// TwinCAT 3 PLC project HardwareSimulator
// ProgramVersion: 3.1.4024.0
// libraries:
//   Tc2_Standard, * (Beckhoff Automation GmbH)
//   Tc2_System, * (Beckhoff Automation GmbH)
//   Tc2_Utilities, * (Beckhoff Automation GmbH)
//   Tc3_Module, * (Beckhoff Automation GmbH)
//   VisuSymbols,3.5.10.0,System
// project tree:
//   / GlobalTextList.TcGTLO (not stored), PlcTask.TcTTO, Visualization Manager.TcVMO (not stored)
//   POUs/ MAIN.TcPOU, SIM_ValveWithFB.TcPOU, SIM_ValveWithDoubleFB.TcPOU, SIM_MOVITRAC_B.TcPOU, SIM_SpeedDoor.TcPOU
//   VISUs/ Visualization.TcVIS
// (motion and I/O tree: see PLC project cleanroomconnect)
// real-time tasks:
//   TASK PlcTask: cycle T#10ms, priority 20, ADS port 350
//   TASK PlcTaskHwSim: cycle T#10ms, priority 21, ADS port 351
// variable links:

CONFIGURATION HardwareSimulator
    RESOURCE PLC ON TwinCAT3
        TASK PlcTask(INTERVAL := T#10ms, PRIORITY := 21);
        PROGRAM MAIN WITH PlcTask : MAIN;
    END_RESOURCE
END_CONFIGURATION

// ---- POUs/MAIN.TcPOU
PROGRAM MAIN
VAR
	//EM Pallet Transport
	simMOVITRAC_B : SIM_MOVITRAC_B;
	simCentering : SIM_ValveWithDoubleFB;
	
	//EM Docking Interface
	simDockingClampUpper : SIM_ValveWithDoubleFB;
	simDockingClampLower : SIM_ValveWithDoubleFB;
	simUnlockPinUpper : SIM_ValveWithFB;
	simUnlockPinLower : SIM_ValveWithFB;
	simDoorOpener : SIM_ValveWithFB;
	simDoorShutter : SIM_ValveWithFB;
	simDoorOpenerAlmostClosed AT %Q* : BOOL;
	tonDoorOpenerAlmosClosed : TON;
	
	//EM Lifting Transport
 	//Via NC-Task
	
	//EM Doors
	simOuterCabinDoor : SIM_SpeedDoor;
	simInnerCabinDoor : SIM_SpeedDoor;
	
	//Safety
	bInitDone : BOOL;
	simSafetyOK AT %Q* : BOOL;
	simPower400VacOK AT %Q* : BOOL;
	simPower230VacOK AT %Q* : BOOL;
	simPower230VacSocketsOK AT %Q* : BOOL;
	simPower48VdcOK AT %Q* : BOOL;
	simPowerPotentialGroupOK AT %Q* : BOOL;
	simAirPressureOK AT %Q* : BOOL;
	simCabinetTemperatureOK AT %Q* : BOOL;
	
	simLiftEnable AT %Q* : BOOL;
	simLiftLimitPos AT %Q* : BOOL;
	simLiftLimitNeg AT %Q* : BOOL;
	simTransportEnable AT %Q* : BOOL;
	simTransportLimitPos AT %Q* : BOOL;
	simTransportLimitNeg AT %Q* : BOOL;
END_VAR


IF NOT(bInitDone) THEN
	simSafetyOK := TRUE;
	simPower400VacOK := TRUE;
	simPower230VacOK := TRUE;
	simPower230VacSocketsOK := TRUE;
	simPower48VdcOK := TRUE;
	simPowerPotentialGroupOK := TRUE;
	simAirPressureOK := TRUE;
	simCabinetTemperatureOK := TRUE;
	
	simLiftEnable := TRUE;
	simLiftLimitPos := TRUE;
	simLiftLimitNeg := TRUE;
	simTransportEnable := TRUE;
	simTransportLimitPos := TRUE;
	simTransportLimitNeg := TRUE;
	
	simDoorShutter.mForceOff();
	simDoorOpener.mForceOff();
	
	bInitDone := TRUE;
END_IF

//EM Pallet Conveyor
simMOVITRAC_B();

simCentering();

//EM Docking Interface
simDockingClampUpper();
simDockingClampLower();
simUnlockPinUpper();
simUnlockPinLower();
simDoorOpener();
simDoorShutter();

tonDoorOpenerAlmosClosed(IN := (simDoorOpener.q_bCmdValveOff OR simDoorOpener.q_bStaValveOff), PT := T#1S);
simDoorOpenerAlmostClosed := tonDoorOpenerAlmosClosed.Q; 

//EM Doors
simOuterCabinDoor();
simInnerCabinDoor();

END_PROGRAM

// ---- POUs/SIM_MOVITRAC_B.TcPOU
FUNCTION_BLOCK SIM_MOVITRAC_B
VAR 
	//Outputs from PLC --> HW
	I_bCmdReset AT %I* : BOOL;
	I_bCmdEnable AT %I* : BOOL;
	I_bCmdStartCW AT %I* : BOOL;
	I_bCmdStartCCW AT %I* : BOOL;
	
	//Inputs from HW --> PLC
	Q_bStaReadyForOperation AT %Q* : BOOL;
	Q_bStaMotorIsRunning AT %Q* : BOOL;
	
	s_tonEnabled : TON;
	s_tonRunning : TON;
	s_tonStopped : TON;
	
	s_bError : BOOL := TRUE;
END_VAR


IF I_bCmdEnable THEN ; END_IF

s_tonEnabled(IN := (*I_bCmdEnable AND*) NOT(s_bError), PT := T#2S);
s_tonRunning(IN := s_tonEnabled.Q AND (I_bCmdStartCW OR I_bCmdStartCCW) , PT := T#2S);
s_tonStopped(IN := NOT(s_tonRunning.Q), PT := T#2S);

Q_bStaReadyForOperation := s_tonEnabled.Q;
Q_bStaMotorIsRunning := s_tonRunning.Q OR NOT(s_tonStopped.Q);

IF I_bCmdReset THEN
	s_bError := FALSE;
END_IF

END_FUNCTION_BLOCK

// ---- POUs/SIM_ValveWithDoubleFB.TcPOU
FUNCTION_BLOCK SIM_ValveWithDoubleFB
VAR 
	//Outputs from PLC --> HW
	I_bCmdValveOn AT %I* : BOOL;
	I_bCmdValveOff AT %I* : BOOL;
	
	//Inputs from HW --> PLC
	Q_bStaFeedbackOn AT %Q* : BOOL;
	Q_bStaFeedbackOff AT %Q* : BOOL;
	Q_bStaFeedbackOn2 AT %Q* : BOOL;
	Q_bStaFeedbackOff2 AT %Q* : BOOL;
	
	s_tonOn : TON;
	s_tonOff : TON;
	
END_VAR

VAR_OUTPUT
	q_bStaValveOn : BOOL;
	q_bStaValveOff : BOOL;
END_VAR


s_tonOn(IN := I_bCmdValveOn AND NOT(I_bCmdValveOff), PT := T#2S);

IF s_tonOn.Q THEN
	Q_bStaFeedbackOn := TRUE;
	Q_bStaFeedbackOn2 := TRUE;
ELSIF I_bCmdValveOff THEN
	Q_bStaFeedbackOn := FALSE;
	Q_bStaFeedbackOn2 := FALSE;
END_IF

s_tonOff(IN := I_bCmdValveOff AND NOT(I_bCmdValveOn), PT := T#2S);

IF s_tonOff.Q THEN
	Q_bStaFeedbackOff := TRUE;
	Q_bStaFeedbackOff2 := TRUE;
ELSIF I_bCmdValveOn THEN
	Q_bStaFeedbackOff := FALSE;
	Q_bStaFeedbackOff2 := FALSE;
END_IF

q_bStaValveOn := Q_bStaFeedbackOn;
q_bStaValveOff := Q_bStaFeedbackOff;

END_FUNCTION_BLOCK

// ---- POUs/SIM_ValveWithFB.TcPOU
FUNCTION_BLOCK SIM_ValveWithFB
VAR
	//Outputs from PLC --> HW
	I_bCmdValveOn AT %I* : BOOL;
	I_bCmdValveOff AT %I* : BOOL;
	
	//Inputs from HW --> PLC
	Q_bStaFeedbackOn AT %Q* : BOOL;
	Q_bStaFeedbackOff AT %Q* : BOOL;
	
	s_tonOn : TON;
	s_tonOff : TON;
	
END_VAR

VAR_OUTPUT
	q_bStaValveOn : BOOL;
	q_bStaValveOff : BOOL;
	
	q_bCmdValveOn : BOOL;	//Q*
	q_bCmdValveOff : BOOL;	//Q*
END_VAR


s_tonOn(IN := I_bCmdValveOn AND NOT(I_bCmdValveOff), PT := T#2S);

IF s_tonOn.Q THEN
	Q_bStaFeedbackOn := TRUE;
ELSIF I_bCmdValveOff THEN
	Q_bStaFeedbackOn := FALSE;
END_IF

s_tonOff(IN := I_bCmdValveOff AND NOT(I_bCmdValveOn), PT := T#2S);

IF s_tonOff.Q THEN
	Q_bStaFeedbackOff := TRUE;
ELSIF I_bCmdValveOn THEN
	Q_bStaFeedbackOff := FALSE;
END_IF

q_bStaValveOn := Q_bStaFeedbackOn;
q_bStaValveOff := Q_bStaFeedbackOff;

q_bCmdValveOn := I_bCmdValveOn;
q_bCmdValveOff := I_bCmdValveOff;

METHOD mForceOff : BOOL

Q_bStaFeedbackOff := TRUE;
END_METHOD

METHOD mForceOn : BOOL

Q_bStaFeedbackOn := TRUE;
END_METHOD

END_FUNCTION_BLOCK

// ---- POUs/SIM_SpeedDoor.TcPOU
FUNCTION_BLOCK SIM_SpeedDoor
VAR
	//Outputs from PLC --> HW
	I_bCmdReset AT %I* : BOOL;
	I_bCmdDoorOpen AT %I* : BOOL;
	I_bCmdDoorClose AT %I* : BOOL;
	
	//Inputs from HW --> PLC
	Q_bStaDoorIsReady AT %Q* : BOOL;
	Q_bStaDoorIsOpened AT %Q* : BOOL;
	Q_bStaDoorIsClosed AT %Q* : BOOL;
	
	s_bCmdOpen : BOOL := FALSE;
	s_bCmdClose : BOOL := TRUE;
	
	s_tonOpen : TON;
	s_tonClose : TON;
	
END_VAR

VAR_OUTPUT
	q_bStaDoorOpen : BOOL;
	q_bStaDoorClose : BOOL;
	
	q_bCmdDoorOpen : BOOL;	//Q*
	q_bCmdDoorClose : BOOL;	//Q*
END_VAR


IF I_bCmdDoorOpen THEN
	s_bCmdOpen := TRUE;
	s_bCmdClose := FALSE;
ELSIF I_bCmdDoorClose THEN
	s_bCmdOpen := FALSE;
	s_bCmdClose := TRUE;
END_IF

s_tonOpen(IN := s_bCmdOpen, PT := T#2S);

IF s_tonOpen.Q THEN
	Q_bStaDoorIsOpened := TRUE;
//ELSIF I_bCmdDoorClose THEN
ELSIF s_bCmdClose THEN
	Q_bStaDoorIsOpened := FALSE;
END_IF
	
s_tonClose(IN := s_bCmdClose, PT := T#2S);

IF s_tonClose.Q THEN
	Q_bStaDoorIsClosed := TRUE;
ELSIF s_bCmdOpen THEN
	Q_bStaDoorIsClosed := FALSE;
END_IF

IF I_bCmdReset THEN
	Q_bStaDoorIsReady := TRUE;
END_IF

q_bStaDoorOpen := Q_bStaDoorIsOpened;
q_bStaDoorClose := Q_bStaDoorIsClosed;

q_bCmdDoorOpen := I_bCmdDoorOpen;
q_bCmdDoorClose := I_bCmdDoorClose;

END_FUNCTION_BLOCK

// ---- VISUs/Visualization.TcVIS
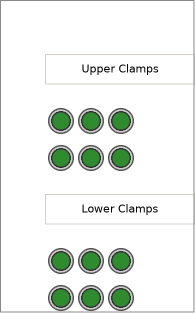
VISUALIZATION Visualization  // 195x313
    Lamp1 (46,106 30x30), variable: MAIN.simClampUpper.I_bCmdValveOff, style: Lamp-Lamp1-Green
    Textfield (45,54 150x30), "Upper Clamps"
    Lamp1 (46,143 30x30), variable: MAIN.simClampUpper.I_bCmdValveOn, style: Lamp-Lamp1-Green
    Lamp1 (76,143 30x30), variable: MAIN.simClampUpper.Q_bStaFeedbackOn, style: Lamp-Lamp1-Green
    Lamp1 (76,106 30x30), variable: MAIN.simClampUpper.Q_bStaFeedbackOff, style: Lamp-Lamp1-Green
    Lamp1 (106,106 30x30), variable: MAIN.simClampUpper.Q_bStaFeedbackOff2, style: Lamp-Lamp1-Green
    Lamp1 (106,143 30x30), variable: MAIN.simClampUpper.Q_bStaFeedbackOn2, style: Lamp-Lamp1-Green
    Lamp1 (46,246 30x30), variable: MAIN.simClampLower.I_bCmdValveOff, style: Lamp-Lamp1-Green
    Textfield (45,194 150x30), "Lower Clamps"
    Lamp1 (46,283 30x30), variable: MAIN.simClampLower.I_bCmdValveOn, style: Lamp-Lamp1-Green
    Lamp1 (76,283 30x30), variable: MAIN.simClampLower.Q_bStaFeedbackOn, style: Lamp-Lamp1-Green
    Lamp1 (76,246 30x30), variable: MAIN.simClampLower.Q_bStaFeedbackOff, style: Lamp-Lamp1-Green
    Lamp1 (106,246 30x30), variable: MAIN.simClampLower.Q_bStaFeedbackOff2, style: Lamp-Lamp1-Green
    Lamp1 (106,283 30x30), variable: MAIN.simClampLower.Q_bStaFeedbackOn2, style: Lamp-Lamp1-Green
END_VISUALIZATION
